// TIA Portal V20 export
FUNCTION_BLOCK "Pallet_Transport_Row_4"   // FB14, LAD
{ S7_Optimized_Access := 'TRUE' }
// stored: MemoryReserve 100, SetENOAutomatically false
   VAR_INPUT
      Start_Station : "Station";
      Destination_Station : "Station";
      Reverse_Rotation : Bool;
      iButton_StS_StD : Bool;
      iButton_StD_StS : Bool;
      isEndingStation_STD : Bool;
      isEndingStation_STS : Bool;
      TandemOperation : Bool;
      TandemSpeed : Int;
   END_VAR
   VAR_OUTPUT
      oButton_StS_StD_LED : Bool;
      oStatus_HMI_StS_StD : Bool;
      oStatus_HMI_StD_StS : Bool;
      oCentering : Bool;
      Stop_Drive_Button : Bool;
      Stop_Drive_HMI : Bool;
      Centering_Alarm : Bool;
   END_VAR
   VAR_IN_OUT
      iDriveStS_Param : "SEW_MOVIKIT_VelocityDrive_SETPOINTS_V2.1";
      oDriveStS_Param : "SEW_MOVIKIT_VelocityDrive_STATUS_V2.1";
      iDriveStD_Param : "SEW_MOVIKIT_VelocityDrive_SETPOINTS_V2.1";
      oDriveStD_Param : "SEW_MOVIKIT_VelocityDrive_STATUS_V2.1";
      iDriveStS_double_Param : "SEW_MOVIKIT_VelocityDrive_SETPOINTS_V2.1";
      oDriveStS_double_Param : "SEW_MOVIKIT_VelocityDrive_STATUS_V2.1";
      iDriveStD_double_Param : "SEW_MOVIKIT_VelocityDrive_SETPOINTS_V2.1";
      oDriveStD_double_Param : "SEW_MOVIKIT_VelocityDrive_STATUS_V2.1";
      isCentering : Bool;
      HMI_StS_StD : Bool;
      HMI_StD_StS : Bool;
   END_VAR
   VAR
      Drive_To_Destination : Bool;
      Set_Speed : Int;
      Set_Speed_Reverse : Int;
      CommunicationOk : Bool;
      Jog_StS : Bool;
      Jog_StD : Bool;
      CenteringStep : Int;
      TON_Centering : TON_TIME;
      trigTimeout { S7_SetPoint := 'True'} : R_TRIG;
      Trig_StS_StD { S7_SetPoint := 'True'} : Bool;
      Trig_StD_StS : Bool;
      Reset_StS_StD : Bool;
      Reset_StD_StS : Bool;
      Timer_Drive_Error_Button : TON_TIME;
      Timer_Drive_Error_HMI : TON_TIME;
      STOP_DRIVERS { S7_SetPoint := 'True'} : Bool;
   END_VAR
   VAR_TEMP
      LED_StD_STS : Bool;
      LED_StS_STD : Bool;
   END_VAR
   VAR CONSTANT
      ACC : Int := 300;
      DCC : Int := 400;
      SPEED_BACK : Int := -100;
      SPEED_FWD : Int := 100;
   END_VAR
   VAR_TEMP   // added for the SCL form of the ladder/FBD networks
      _w1 : Bool;
      _w2 : Bool;
      _w3 : Bool;
      _w4 : Bool;
   END_VAR
BEGIN

REGION Network 1: Reset commands
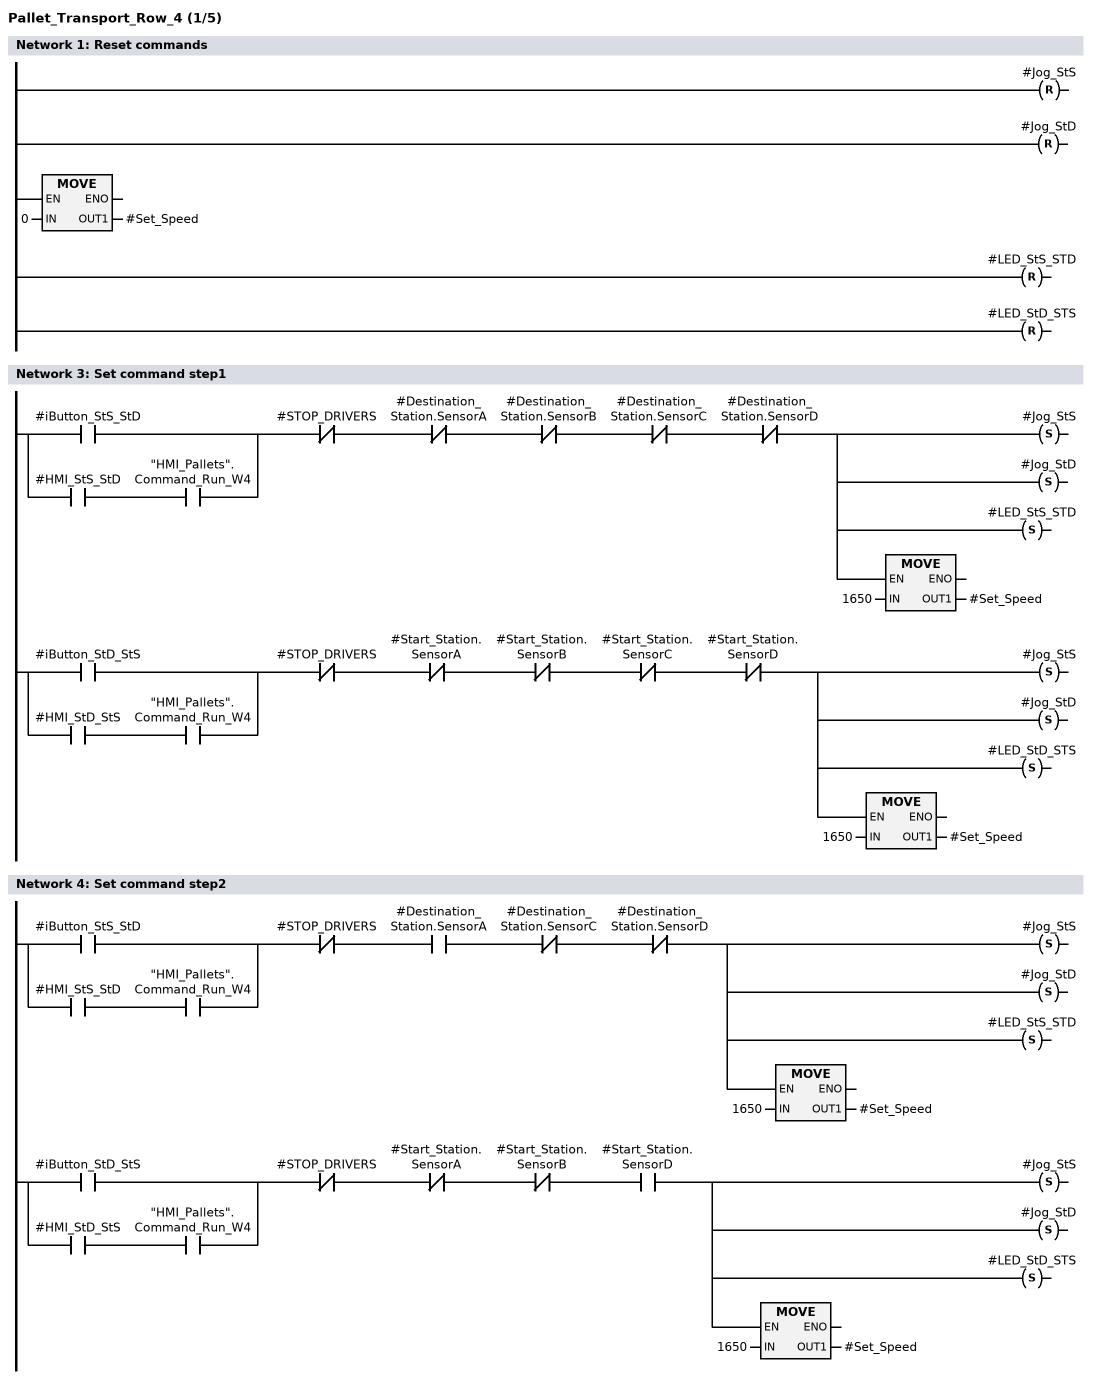
   RUNG wire#powerrail
      R_Coil( #Jog_StS )
   END_RUNG
   RUNG wire#powerrail
      R_Coil( #Jog_StD )
   END_RUNG
   RUNG wire#powerrail
      Move(in := 0, out1 => #Set_Speed)
   END_RUNG
   RUNG wire#powerrail
      R_Coil( #LED_StS_STD )
   END_RUNG
   RUNG wire#powerrail
      R_Coil( #LED_StD_STS )
   END_RUNG
   // the same network as SCL:
   #Jog_StS := FALSE;
   #Jog_StD := FALSE;
   #Set_Speed := 0;
   #LED_StS_STD := FALSE;
   #LED_StD_STS := FALSE;
END_REGION

REGION Network 2 (SCL): Triggers STOP_DRIVERS after 8 s of active move command without motion
   #Timer_Drive_Error_Button(
                             IN :=
                             (
                             #iButton_StS_StD OR
                             #iButton_StD_StS
                             )
                             AND NOT (
                             #oDriveStS_Param.x_Bit_4_Motor_turning OR
                             #oDriveStS_double_Param.x_Bit_4_Motor_turning OR
                             #oDriveStD_Param.x_Bit_4_Motor_turning OR
                             #oDriveStD_double_Param.x_Bit_4_Motor_turning
                             ),
                             PT := T#15s
   );


   #Timer_Drive_Error_HMI(
                          IN :=
                          (
                          #HMI_StS_StD OR
                          #HMI_StD_StS
                          )
                          AND NOT (
                          #oDriveStS_Param.x_Bit_4_Motor_turning OR
                          #oDriveStS_double_Param.x_Bit_4_Motor_turning OR
                          #oDriveStD_Param.x_Bit_4_Motor_turning OR
                          #oDriveStD_double_Param.x_Bit_4_Motor_turning
                          ),
                          PT := T#10s
   );

   IF #Timer_Drive_Error_Button.Q THEN
       #STOP_DRIVERS := TRUE;
       #Stop_Drive_Button := TRUE;
   END_IF;


   IF #Timer_Drive_Error_HMI.Q THEN
       #STOP_DRIVERS := TRUE;
       #Stop_Drive_HMI := TRUE;
       #HMI_StS_StD := FALSE;
       #HMI_StD_StS := FALSE;
   END_IF;


   IF "HMI_Pallets".Reset_Drivers THEN
       #STOP_DRIVERS := FALSE;
       #Stop_Drive_Button := FALSE;
       #Stop_Drive_HMI := FALSE;
   END_IF;
END_REGION

REGION Network 3: Set command step1
   RUNG wire#powerrail
      Contact( #iButton_StS_StD )
      wire#w1
      I_Contact( #STOP_DRIVERS )
      I_Contact( #Destination_Station.SensorA )
      I_Contact( #Destination_Station.SensorB )
      I_Contact( #Destination_Station.SensorC )
      I_Contact( #Destination_Station.SensorD )
      wire#w2
      S_Coil( #Jog_StS )
   END_RUNG
   RUNG wire#powerrail
      Contact( #HMI_StS_StD )
      Contact( "HMI_Pallets".Command_Run_W4 )
   END_RUNG wire#w1
   RUNG wire#w2
      S_Coil( #Jog_StD )
   END_RUNG
   RUNG wire#w2
      S_Coil( #LED_StS_STD )
   END_RUNG
   RUNG wire#w2
      Move(in := 1650, out1 => #Set_Speed)
   END_RUNG
   RUNG wire#powerrail
      Contact( #iButton_StD_StS )
      wire#w3
      I_Contact( #STOP_DRIVERS )
      I_Contact( #Start_Station.SensorA )
      I_Contact( #Start_Station.SensorB )
      I_Contact( #Start_Station.SensorC )
      I_Contact( #Start_Station.SensorD )
      wire#w4
      S_Coil( #Jog_StS )
   END_RUNG
   RUNG wire#powerrail
      Contact( #HMI_StD_StS )
      Contact( "HMI_Pallets".Command_Run_W4 )
   END_RUNG wire#w3
   RUNG wire#w4
      S_Coil( #Jog_StD )
   END_RUNG
   RUNG wire#w4
      S_Coil( #LED_StD_STS )
   END_RUNG
   RUNG wire#w4
      Move(in := 1650, out1 => #Set_Speed)
   END_RUNG
   // the same network as SCL:
   IF (#iButton_StS_StD OR (#HMI_StS_StD AND "HMI_Pallets".Command_Run_W4)) AND NOT #STOP_DRIVERS AND NOT #Destination_Station.SensorA AND NOT #Destination_Station.SensorB AND NOT #Destination_Station.SensorC AND NOT #Destination_Station.SensorD THEN
       #Jog_StS := TRUE;
       #Jog_StD := TRUE;
       #LED_StS_STD := TRUE;
       #Set_Speed := 1650;
   END_IF;
   IF (#iButton_StD_StS OR (#HMI_StD_StS AND "HMI_Pallets".Command_Run_W4)) AND NOT #STOP_DRIVERS AND NOT #Start_Station.SensorA AND NOT #Start_Station.SensorB AND NOT #Start_Station.SensorC AND NOT #Start_Station.SensorD THEN
       #Jog_StS := TRUE;
       #Jog_StD := TRUE;
       #LED_StD_STS := TRUE;
       #Set_Speed := 1650;
   END_IF;
END_REGION

REGION Network 4: Set command step2
   RUNG wire#powerrail
      Contact( #iButton_StS_StD )
      wire#w1
      I_Contact( #STOP_DRIVERS )
      Contact( #Destination_Station.SensorA )
      I_Contact( #Destination_Station.SensorC )
      I_Contact( #Destination_Station.SensorD )
      wire#w2
      S_Coil( #Jog_StS )
   END_RUNG
   RUNG wire#powerrail
      Contact( #HMI_StS_StD )
      Contact( "HMI_Pallets".Command_Run_W4 )
   END_RUNG wire#w1
   RUNG wire#w2
      S_Coil( #Jog_StD )
   END_RUNG
   RUNG wire#w2
      S_Coil( #LED_StS_STD )
   END_RUNG
   RUNG wire#w2
      Move(in := 1650, out1 => #Set_Speed)
   END_RUNG
   RUNG wire#powerrail
      Contact( #iButton_StD_StS )
      wire#w3
      I_Contact( #STOP_DRIVERS )
      I_Contact( #Start_Station.SensorA )
      I_Contact( #Start_Station.SensorB )
      Contact( #Start_Station.SensorD )
      wire#w4
      S_Coil( #Jog_StS )
   END_RUNG
   RUNG wire#powerrail
      Contact( #HMI_StD_StS )
      Contact( "HMI_Pallets".Command_Run_W4 )
   END_RUNG wire#w3
   RUNG wire#w4
      S_Coil( #Jog_StD )
   END_RUNG
   RUNG wire#w4
      S_Coil( #LED_StD_STS )
   END_RUNG
   RUNG wire#w4
      Move(in := 1650, out1 => #Set_Speed)
   END_RUNG
   // the same network as SCL:
   IF (#iButton_StS_StD OR (#HMI_StS_StD AND "HMI_Pallets".Command_Run_W4)) AND NOT #STOP_DRIVERS AND #Destination_Station.SensorA AND NOT #Destination_Station.SensorC AND NOT #Destination_Station.SensorD THEN
       #Jog_StS := TRUE;
       #Jog_StD := TRUE;
       #LED_StS_STD := TRUE;
       #Set_Speed := 1650;
   END_IF;
   IF (#iButton_StD_StS OR (#HMI_StD_StS AND "HMI_Pallets".Command_Run_W4)) AND NOT #STOP_DRIVERS AND NOT #Start_Station.SensorA AND NOT #Start_Station.SensorB AND #Start_Station.SensorD THEN
       #Jog_StS := TRUE;
       #Jog_StD := TRUE;
       #LED_StD_STS := TRUE;
       #Set_Speed := 1650;
   END_IF;
END_REGION

REGION Network 5: Set command step3
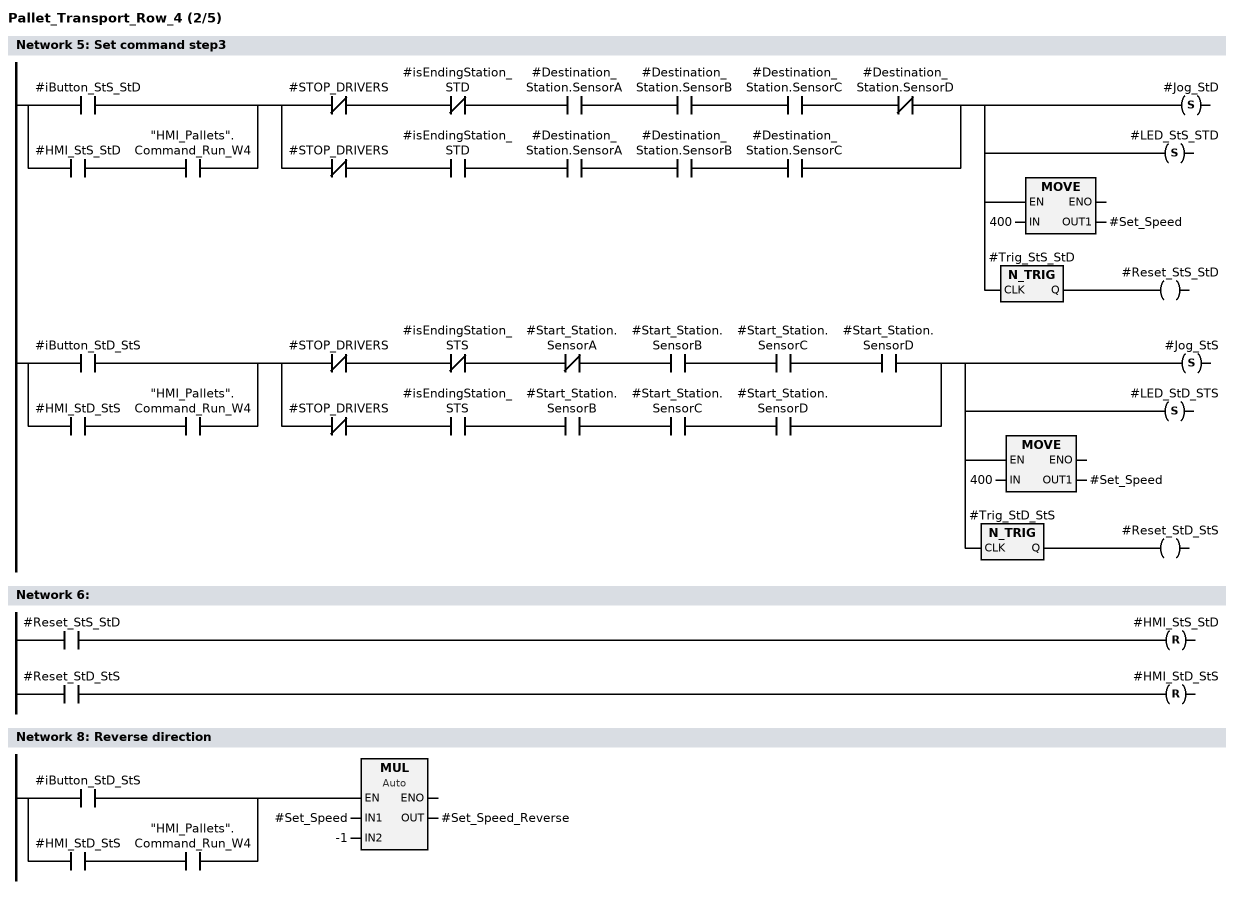
   RUNG wire#powerrail
      Contact( #iButton_StS_StD )
      wire#w1
      I_Contact( #STOP_DRIVERS )
      I_Contact( #isEndingStation_STD )
      Contact( #Destination_Station.SensorA )
      Contact( #Destination_Station.SensorB )
      Contact( #Destination_Station.SensorC )
      I_Contact( #Destination_Station.SensorD )
      wire#w2
      S_Coil( #Jog_StD )
   END_RUNG
   RUNG wire#powerrail
      Contact( #HMI_StS_StD )
      Contact( "HMI_Pallets".Command_Run_W4 )
   END_RUNG wire#w1
   RUNG wire#w1
      I_Contact( #STOP_DRIVERS )
      Contact( #isEndingStation_STD )
      Contact( #Destination_Station.SensorA )
      Contact( #Destination_Station.SensorB )
      Contact( #Destination_Station.SensorC )
   END_RUNG wire#w2
   RUNG wire#w2
      S_Coil( #LED_StS_STD )
   END_RUNG
   RUNG wire#w2
      Move(in := 400, out1 => #Set_Speed)
   END_RUNG
   RUNG wire#w2
      N_Trig( #Trig_StS_StD )
      Coil( #Reset_StS_StD )
   END_RUNG
   RUNG wire#powerrail
      Contact( #iButton_StD_StS )
      wire#w3
      I_Contact( #STOP_DRIVERS )
      I_Contact( #isEndingStation_STS )
      I_Contact( #Start_Station.SensorA )
      Contact( #Start_Station.SensorB )
      Contact( #Start_Station.SensorC )
      Contact( #Start_Station.SensorD )
      wire#w4
      S_Coil( #Jog_StS )
   END_RUNG
   RUNG wire#powerrail
      Contact( #HMI_StD_StS )
      Contact( "HMI_Pallets".Command_Run_W4 )
   END_RUNG wire#w3
   RUNG wire#w3
      I_Contact( #STOP_DRIVERS )
      Contact( #isEndingStation_STS )
      Contact( #Start_Station.SensorB )
      Contact( #Start_Station.SensorC )
      Contact( #Start_Station.SensorD )
   END_RUNG wire#w4
   RUNG wire#w4
      S_Coil( #LED_StD_STS )
   END_RUNG
   RUNG wire#w4
      Move(in := 400, out1 => #Set_Speed)
   END_RUNG
   RUNG wire#w4
      N_Trig( #Trig_StD_StS )
      Coil( #Reset_StD_StS )
   END_RUNG
   // the same network as SCL:
   #_w1 := (#iButton_StS_StD OR (#HMI_StS_StD AND "HMI_Pallets".Command_Run_W4)) AND ((NOT #STOP_DRIVERS AND NOT #isEndingStation_STD AND #Destination_Station.SensorA AND #Destination_Station.SensorB AND #Destination_Station.SensorC AND NOT #Destination_Station.SensorD) OR (NOT #STOP_DRIVERS AND #isEndingStation_STD AND #Destination_Station.SensorA AND #Destination_Station.SensorB AND #Destination_Station.SensorC));
   IF #_w1 THEN
       #Jog_StD := TRUE;
       #LED_StS_STD := TRUE;
       #Set_Speed := 400;
   END_IF;
   #_w2 := NOT #_w1 AND #Trig_StS_StD;   // falling edge
   #Trig_StS_StD := #_w1;
   #Reset_StS_StD := #_w2;
   #_w3 := (#iButton_StD_StS OR (#HMI_StD_StS AND "HMI_Pallets".Command_Run_W4)) AND ((NOT #STOP_DRIVERS AND NOT #isEndingStation_STS AND NOT #Start_Station.SensorA AND #Start_Station.SensorB AND #Start_Station.SensorC AND #Start_Station.SensorD) OR (NOT #STOP_DRIVERS AND #isEndingStation_STS AND #Start_Station.SensorB AND #Start_Station.SensorC AND #Start_Station.SensorD));
   IF #_w3 THEN
       #Jog_StS := TRUE;
       #LED_StD_STS := TRUE;
       #Set_Speed := 400;
   END_IF;
   #_w4 := NOT #_w3 AND #Trig_StD_StS;   // falling edge
   #Trig_StD_StS := #_w3;
   #Reset_StD_StS := #_w4;
END_REGION

REGION Network 6
   RUNG wire#powerrail
      Contact( #Reset_StS_StD )
      R_Coil( #HMI_StS_StD )
   END_RUNG
   RUNG wire#powerrail
      Contact( #Reset_StD_StS )
      R_Coil( #HMI_StD_StS )
   END_RUNG
   // the same network as SCL:
   IF #Reset_StS_StD THEN #HMI_StS_StD := FALSE; END_IF;
   IF #Reset_StD_StS THEN #HMI_StD_StS := FALSE; END_IF;
END_REGION

REGION Network 7 (SCL): Centering
   IF NOT #Destination_Station.SensorB OR
       NOT #Destination_Station.SensorC THEN
       #oCentering := 0;
       #CenteringStep := 0;
       IF #isCentering THEN
           #Centering_Alarm := TRUE;
           #isCentering := FALSE;
       END_IF;
   END_IF;

   IF #isCentering THEN
       CASE #CenteringStep OF
           0:
               IF #Destination_Station.SensorB AND
                   #Destination_Station.SensorC AND
                   #Destination_Station.SensorD THEN
                   #Set_Speed := #SPEED_BACK;
                   //#Jog_StS := TRUE;
                   #Jog_StD := TRUE;
               END_IF;

               IF  #Destination_Station.SensorB AND
                   #Destination_Station.SensorC AND
                   NOT #Destination_Station.SensorD THEN
                   #CenteringStep := 1;
               END_IF;

           1:
               #Set_Speed := #SPEED_FWD;
               //  #Jog_StS := TRUE;
               #Jog_StD := TRUE;
               IF #Destination_Station.SensorD THEN
                   #CenteringStep := 2;
               END_IF;

           2:
               #Set_Speed := 0;
               // #Jog_StS := FALSE;
               #Jog_StD := FALSE;
               #oCentering := TRUE;
               #CenteringStep := 0;
               #isCentering := FALSE;
               #Centering_Alarm := FALSE;
       END_CASE;
   END_IF;

   #TON_Centering(IN := #isCentering,
                  PT := T#8s);

   #trigTimeout(CLK := #TON_Centering.Q);

   // Wykona się tylko raz, gdy minie 8s
   IF #trigTimeout.Q THEN
       #Centering_Alarm := TRUE;
       #isCentering := FALSE;
       #CenteringStep := 0;
       #Set_Speed := 0;
       #Jog_StD := FALSE;
       #Jog_StS := FALSE;
   END_IF;
END_REGION

REGION Network 8: Reverse direction
   RUNG wire#powerrail
      Contact( #iButton_StD_StS )
      wire#w1
      Mul(in1 := #Set_Speed, in2 := -1, out => #Set_Speed_Reverse)
   END_RUNG
   RUNG wire#powerrail
      Contact( #HMI_StD_StS )
      Contact( "HMI_Pallets".Command_Run_W4 )
   END_RUNG wire#w1
   // the same network as SCL:
   IF #iButton_StD_StS OR (#HMI_StD_StS AND "HMI_Pallets".Command_Run_W4) THEN
       #Set_Speed_Reverse := #Set_Speed * (-1);
   END_IF;
END_REGION

REGION Network 9: StS Drive
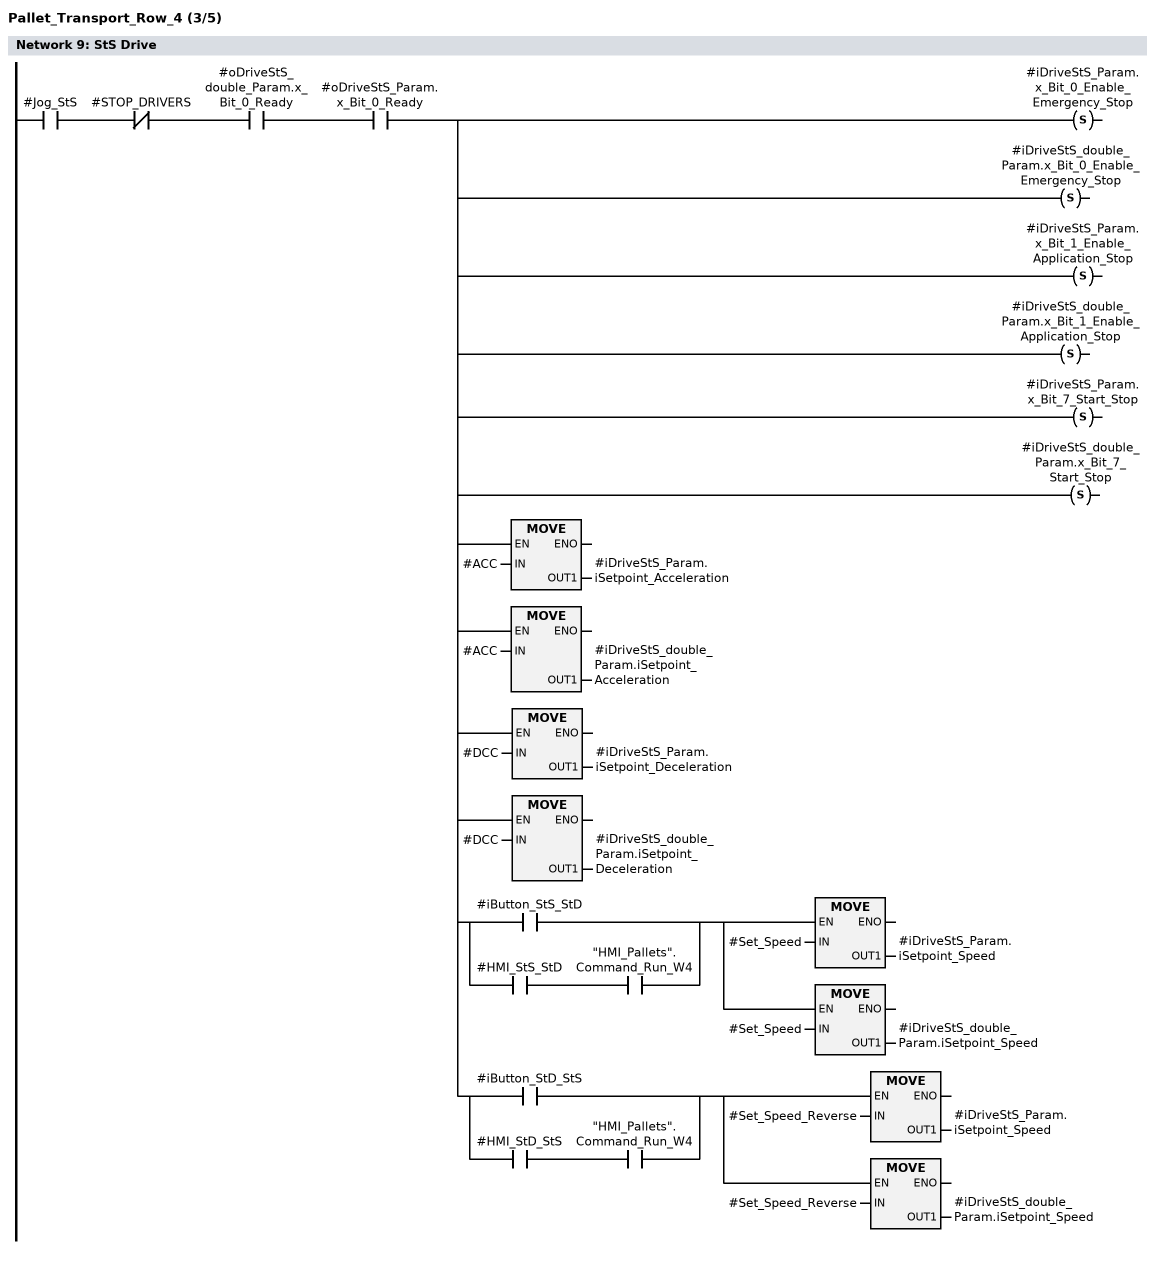
   RUNG wire#powerrail
      Contact( #Jog_StS )
      I_Contact( #STOP_DRIVERS )
      Contact( #oDriveStS_double_Param.x_Bit_0_Ready )
      Contact( #oDriveStS_Param.x_Bit_0_Ready )
      wire#w1
      S_Coil( #iDriveStS_Param.x_Bit_0_Enable_Emergency_Stop )
   END_RUNG
   RUNG wire#w1
      S_Coil( #iDriveStS_double_Param.x_Bit_0_Enable_Emergency_Stop )
   END_RUNG
   RUNG wire#w1
      S_Coil( #iDriveStS_Param.x_Bit_1_Enable_Application_Stop )
   END_RUNG
   RUNG wire#w1
      S_Coil( #iDriveStS_double_Param.x_Bit_1_Enable_Application_Stop )
   END_RUNG
   RUNG wire#w1
      S_Coil( #iDriveStS_Param.x_Bit_7_Start_Stop )
   END_RUNG
   RUNG wire#w1
      S_Coil( #iDriveStS_double_Param.x_Bit_7_Start_Stop )
   END_RUNG
   RUNG wire#w1
      Move(in := #ACC, out1 => #iDriveStS_Param.iSetpoint_Acceleration)
   END_RUNG
   RUNG wire#w1
      Move(in := #ACC, out1 => #iDriveStS_double_Param.iSetpoint_Acceleration)
   END_RUNG
   RUNG wire#w1
      Move(in := #DCC, out1 => #iDriveStS_Param.iSetpoint_Deceleration)
   END_RUNG
   RUNG wire#w1
      Move(in := #DCC, out1 => #iDriveStS_double_Param.iSetpoint_Deceleration)
   END_RUNG
   RUNG wire#w1
      Contact( #iButton_StS_StD )
      wire#w2
      Move(in := #Set_Speed, out1 => #iDriveStS_Param.iSetpoint_Speed)
   END_RUNG
   RUNG wire#w1
      Contact( #HMI_StS_StD )
      Contact( "HMI_Pallets".Command_Run_W4 )
   END_RUNG wire#w2
   RUNG wire#w2
      Move(in := #Set_Speed, out1 => #iDriveStS_double_Param.iSetpoint_Speed)
   END_RUNG
   RUNG wire#w1
      Contact( #iButton_StD_StS )
      wire#w3
      Move(in := #Set_Speed_Reverse, out1 => #iDriveStS_Param.iSetpoint_Speed)
   END_RUNG
   RUNG wire#w1
      Contact( #HMI_StD_StS )
      Contact( "HMI_Pallets".Command_Run_W4 )
   END_RUNG wire#w3
   RUNG wire#w3
      Move(in := #Set_Speed_Reverse, out1 => #iDriveStS_double_Param.iSetpoint_Speed)
   END_RUNG
   // the same network as SCL:
   #_w1 := #Jog_StS AND NOT #STOP_DRIVERS AND #oDriveStS_double_Param.x_Bit_0_Ready AND #oDriveStS_Param.x_Bit_0_Ready;
   IF #_w1 THEN
       #iDriveStS_Param.x_Bit_0_Enable_Emergency_Stop := TRUE;
       #iDriveStS_double_Param.x_Bit_0_Enable_Emergency_Stop := TRUE;
       #iDriveStS_Param.x_Bit_1_Enable_Application_Stop := TRUE;
       #iDriveStS_double_Param.x_Bit_1_Enable_Application_Stop := TRUE;
       #iDriveStS_Param.x_Bit_7_Start_Stop := TRUE;
       #iDriveStS_double_Param.x_Bit_7_Start_Stop := TRUE;
       #iDriveStS_Param.iSetpoint_Acceleration := #ACC;
       #iDriveStS_double_Param.iSetpoint_Acceleration := #ACC;
       #iDriveStS_Param.iSetpoint_Deceleration := #DCC;
       #iDriveStS_double_Param.iSetpoint_Deceleration := #DCC;
   END_IF;
   IF #_w1 AND (#iButton_StS_StD OR (#HMI_StS_StD AND "HMI_Pallets".Command_Run_W4)) THEN
       #iDriveStS_Param.iSetpoint_Speed := #Set_Speed;
       #iDriveStS_double_Param.iSetpoint_Speed := #Set_Speed;
   END_IF;
   IF #_w1 AND (#iButton_StD_StS OR (#HMI_StD_StS AND "HMI_Pallets".Command_Run_W4)) THEN
       #iDriveStS_Param.iSetpoint_Speed := #Set_Speed_Reverse;
       #iDriveStS_double_Param.iSetpoint_Speed := #Set_Speed_Reverse;
   END_IF;
END_REGION

REGION Network 10: StC Drive
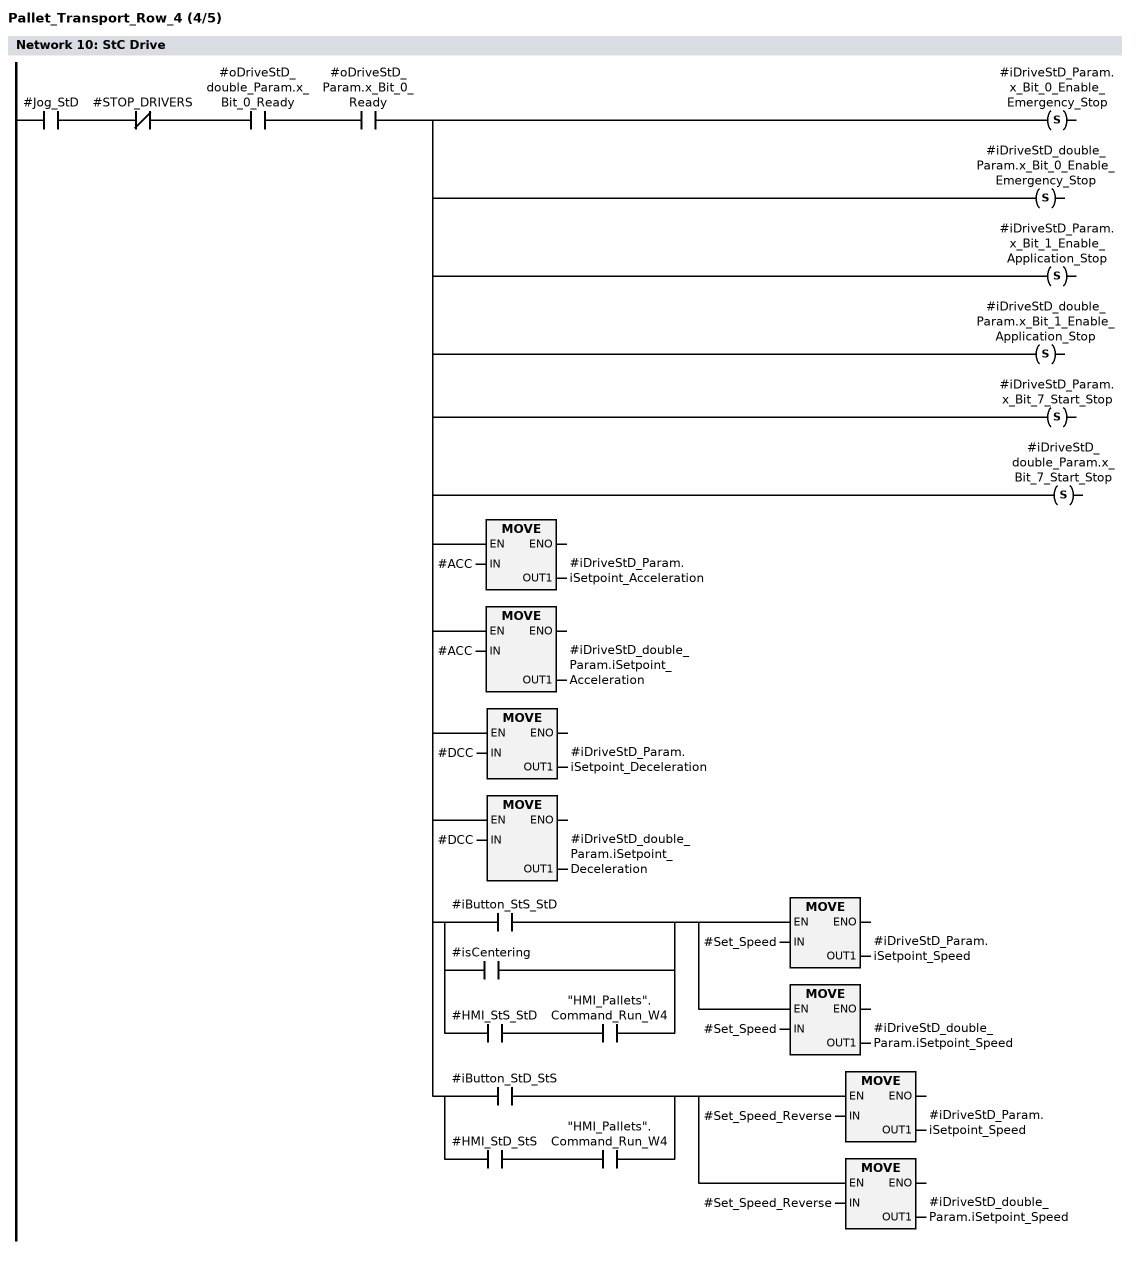
   RUNG wire#powerrail
      Contact( #Jog_StD )
      I_Contact( #STOP_DRIVERS )
      Contact( #oDriveStD_double_Param.x_Bit_0_Ready )
      Contact( #oDriveStD_Param.x_Bit_0_Ready )
      wire#w1
      S_Coil( #iDriveStD_Param.x_Bit_0_Enable_Emergency_Stop )
   END_RUNG
   RUNG wire#w1
      S_Coil( #iDriveStD_double_Param.x_Bit_0_Enable_Emergency_Stop )
   END_RUNG
   RUNG wire#w1
      S_Coil( #iDriveStD_Param.x_Bit_1_Enable_Application_Stop )
   END_RUNG
   RUNG wire#w1
      S_Coil( #iDriveStD_double_Param.x_Bit_1_Enable_Application_Stop )
   END_RUNG
   RUNG wire#w1
      S_Coil( #iDriveStD_Param.x_Bit_7_Start_Stop )
   END_RUNG
   RUNG wire#w1
      S_Coil( #iDriveStD_double_Param.x_Bit_7_Start_Stop )
   END_RUNG
   RUNG wire#w1
      Move(in := #ACC, out1 => #iDriveStD_Param.iSetpoint_Acceleration)
   END_RUNG
   RUNG wire#w1
      Move(in := #ACC, out1 => #iDriveStD_double_Param.iSetpoint_Acceleration)
   END_RUNG
   RUNG wire#w1
      Move(in := #DCC, out1 => #iDriveStD_Param.iSetpoint_Deceleration)
   END_RUNG
   RUNG wire#w1
      Move(in := #DCC, out1 => #iDriveStD_double_Param.iSetpoint_Deceleration)
   END_RUNG
   RUNG wire#w1
      Contact( #iButton_StS_StD )
      wire#w2
      Move(in := #Set_Speed, out1 => #iDriveStD_Param.iSetpoint_Speed)
   END_RUNG
   RUNG wire#w1
      Contact( #isCentering )
   END_RUNG wire#w2
   RUNG wire#w1
      Contact( #HMI_StS_StD )
      Contact( "HMI_Pallets".Command_Run_W4 )
   END_RUNG wire#w2
   RUNG wire#w2
      Move(in := #Set_Speed, out1 => #iDriveStD_double_Param.iSetpoint_Speed)
   END_RUNG
   RUNG wire#w1
      Contact( #iButton_StD_StS )
      wire#w3
      Move(in := #Set_Speed_Reverse, out1 => #iDriveStD_Param.iSetpoint_Speed)
   END_RUNG
   RUNG wire#w1
      Contact( #HMI_StD_StS )
      Contact( "HMI_Pallets".Command_Run_W4 )
   END_RUNG wire#w3
   RUNG wire#w3
      Move(in := #Set_Speed_Reverse, out1 => #iDriveStD_double_Param.iSetpoint_Speed)
   END_RUNG
   // the same network as SCL:
   #_w1 := #Jog_StD AND NOT #STOP_DRIVERS AND #oDriveStD_double_Param.x_Bit_0_Ready AND #oDriveStD_Param.x_Bit_0_Ready;
   IF #_w1 THEN
       #iDriveStD_Param.x_Bit_0_Enable_Emergency_Stop := TRUE;
       #iDriveStD_double_Param.x_Bit_0_Enable_Emergency_Stop := TRUE;
       #iDriveStD_Param.x_Bit_1_Enable_Application_Stop := TRUE;
       #iDriveStD_double_Param.x_Bit_1_Enable_Application_Stop := TRUE;
       #iDriveStD_Param.x_Bit_7_Start_Stop := TRUE;
       #iDriveStD_double_Param.x_Bit_7_Start_Stop := TRUE;
       #iDriveStD_Param.iSetpoint_Acceleration := #ACC;
       #iDriveStD_double_Param.iSetpoint_Acceleration := #ACC;
       #iDriveStD_Param.iSetpoint_Deceleration := #DCC;
       #iDriveStD_double_Param.iSetpoint_Deceleration := #DCC;
   END_IF;
   IF #_w1 AND (#iButton_StS_StD OR #isCentering OR (#HMI_StS_StD AND "HMI_Pallets".Command_Run_W4)) THEN
       #iDriveStD_Param.iSetpoint_Speed := #Set_Speed;
       #iDriveStD_double_Param.iSetpoint_Speed := #Set_Speed;
   END_IF;
   IF #_w1 AND (#iButton_StD_StS OR (#HMI_StD_StS AND "HMI_Pallets".Command_Run_W4)) THEN
       #iDriveStD_Param.iSetpoint_Speed := #Set_Speed_Reverse;
       #iDriveStD_double_Param.iSetpoint_Speed := #Set_Speed_Reverse;
   END_IF;
END_REGION

REGION Network 11: StS -> StD Status
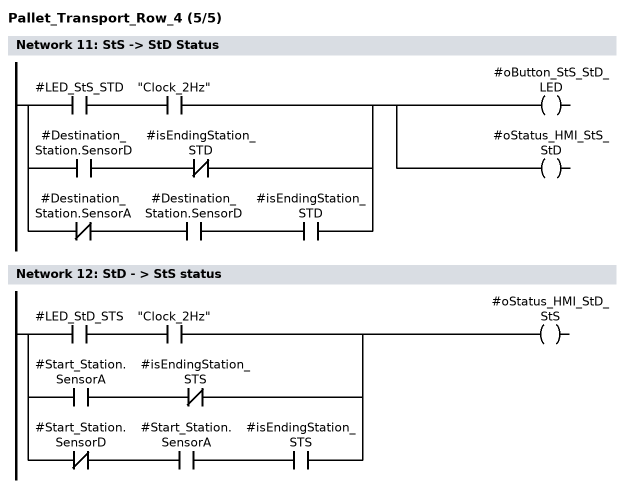
   RUNG wire#powerrail
      Contact( #LED_StS_STD )
      Contact( "Clock_2Hz" )
      wire#w1
      Coil( #oButton_StS_StD_LED )
   END_RUNG
   RUNG wire#powerrail
      Contact( #Destination_Station.SensorD )
      I_Contact( #isEndingStation_STD )
   END_RUNG wire#w1
   RUNG wire#powerrail
      I_Contact( #Destination_Station.SensorA )
      Contact( #Destination_Station.SensorD )
      Contact( #isEndingStation_STD )
   END_RUNG wire#w1
   RUNG wire#w1
      Coil( #oStatus_HMI_StS_StD )
   END_RUNG
   // the same network as SCL:
   #oButton_StS_StD_LED := (#LED_StS_STD AND "Clock_2Hz") OR (#Destination_Station.SensorD AND NOT #isEndingStation_STD) OR (NOT #Destination_Station.SensorA AND #Destination_Station.SensorD AND #isEndingStation_STD);
   #oStatus_HMI_StS_StD := #oButton_StS_StD_LED;
END_REGION

REGION Network 12: StD - > StS status
   RUNG wire#powerrail
      Contact( #LED_StD_STS )
      Contact( "Clock_2Hz" )
      wire#w1
      Coil( #oStatus_HMI_StD_StS )
   END_RUNG
   RUNG wire#powerrail
      Contact( #Start_Station.SensorA )
      I_Contact( #isEndingStation_STS )
   END_RUNG wire#w1
   RUNG wire#powerrail
      I_Contact( #Start_Station.SensorD )
      Contact( #Start_Station.SensorA )
      Contact( #isEndingStation_STS )
   END_RUNG wire#w1
   // the same network as SCL:
   #oStatus_HMI_StD_StS := (#LED_StD_STS AND "Clock_2Hz") OR (#Start_Station.SensorA AND NOT #isEndingStation_STS) OR (NOT #Start_Station.SensorD AND #Start_Station.SensorA AND #isEndingStation_STS);
END_REGION

REGION Network 13 (SCL): Centering status reset
   IF #oCentering AND (#iDriveStD_Param.x_Bit_1_Enable_Application_Stop  OR NOT #Destination_Station.SensorD) THEN
       #oCentering := 0;
   END_IF;
END_REGION
END_FUNCTION_BLOCK
